// TIA Portal V19 export
DATA_BLOCK "PPrgArchive18"   // DB514
// stored: IsOnlyStoredInLoadMemory true, MemoryReserve 0, Namespace G
   VAR RETAIN
      PRG : Array[1701..1800] of "PPrg_Data";
   END_VAR
BEGIN
END_DATA_BLOCK
